Yaskawa INFORM job: KRIS7.JBI

/JOB
//NAME KRIS7
//POS
///NPOS 416,416,416,15,0,0
///TOOL 0
///POSTYPE PULSE
///PULSE
C00000=-36471,-76527,-106813,19264,71481,77238
C00001=-36471,-76527,-106813,19264,71481,77238
C00002=-63812,-119516,-80644,-27282,71106,59809
C00003=-86670,-29465,-24103,-33182,93398,46515
C00004=-88663,-31189,-25266,-33292,92471,45985
C00005=-89600,-31952,-25776,-33339,92036,45737
C00006=-88663,-31189,-25266,-33292,92471,45985
C00007=-88663,-31929,-28188,-33361,93666,45629
C00008=-101397,-33118,-34088,-22474,91022,41668
C00009=-101397,-32934,-33069,-22469,90527,41762
C00010=-101397,-33275,-35023,-22483,91481,41581
C00011=-104499,20623,14787,-23283,115207,62973
C00012=-104352,17765,12486,-23220,115200,63034
C00013=-104529,15851,10717,-23303,115245,62949
C00014=-104352,17765,12486,-23220,115200,63034
C00015=-100086,19810,13187,-22516,115799,63398
C00016=-93288,781,-1160,-33549,91987,44264
C00017=-95103,1586,-482,-33591,91265,43744
C00018=-95638,1156,-842,-33600,91054,43591
C00019=-95103,1586,-482,-33591,91265,43744
C00020=-100253,-3614,-11898,-25466,91372,41970
C00021=-107199,-8537,-17665,-19004,89460,40114
C00022=-108350,-8919,-17473,-17740,88760,39873
C00023=-102096,-5783,-13006,-25389,90415,41488
C00024=-93175,-13453,-24658,-25770,96080,43586
C00025=-29596,-126908,-80456,-16683,91164,67663
C00026=-130966,-130992,-81417,14801,93022,-34731
C00027=-139735,-123676,-71676,23223,79574,-40827
C00028=-136755,-124231,-71804,23689,78586,-39979
C00029=-134984,-124514,-71869,23951,78010,-39473
C00030=-136755,-124231,-71804,23689,78586,-39979
C00031=-136306,-124758,-74432,23664,79703,-39597
C00032=-105195,-127447,-79852,15126,73259,-28242
C00033=-104798,-126140,-77647,15190,72530,-28198
C00034=-108375,-128078,-79564,15067,73342,-29336
C00035=-112121,-93277,-65445,16297,96104,-47809
C00036=-116095,-84503,-58814,18813,102506,-48434
C00037=-114391,-86924,-59797,19239,101506,-47972
C00038=-116095,-84503,-58814,18813,102506,-48434
C00039=-117812,-129995,-81150,14641,74986,-32390
C00040=-118791,-92886,-67151,14205,85296,-31516
C00041=-116748,-92781,-67110,14299,84968,-30842
C00042=-115499,-92681,-67072,14351,84774,-30431
C00043=-116748,-92781,-67110,14299,84968,-30842
C00044=-116748,-94243,-70296,14285,86141,-30707
C00045=-102870,-92009,-70676,9222,86435,-25689
C00046=-102870,-90997,-68303,9229,85506,-25758
C00047=-102870,-92009,-70676,9222,86435,-25689
C00048=-124106,-98193,-79828,8318,91183,-32632
C00049=-120990,-117719,-86799,1028,78019,83969
C00050=-103618,-122878,-84450,6731,45671,69045
C00051=-107839,-39273,-43881,11021,86771,60654
C00052=-102663,-26959,-34255,5037,90909,61236
C00053=-106417,-22492,-30421,10624,98396,60708
C00054=-103076,-37240,-40581,8849,97261,61678
C00055=-110992,-39766,-43585,17340,97602,59383
C00056=-111851,-103912,-94699,10334,87868,68255
C00057=-100525,-93554,-87313,9422,87254,72087
C00058=-95765,-72558,-76889,7644,100510,59309
C00059=-95463,-76426,-71939,16938,115118,61391
C00060=-102124,-64154,-61473,23072,122501,60539
C00061=-108072,-63754,-61449,27079,123073,58329
C00062=-126453,-110744,-88068,25157,96958,85114
C00063=-124535,-114305,-86499,25277,93833,85163
C00064=-121951,-112497,-85625,25654,93398,86032
C00065=-116232,-108405,-84002,26384,92604,88006
C00066=-122754,-106725,-87203,25770,97209,86568
C00067=-142865,-91008,-85242,17891,113758,73123
C00068=-142005,-90205,-84914,18160,113770,73464
C00069=-93871,-48257,-54590,-14207,101968,-48555
C00070=-106716,17042,-5346,-15024,102835,-53222
C00071=-114740,-14345,-34597,-13608,101053,-59815
C00072=-127078,-3386,-21930,-8482,103399,-53955
C00073=-129021,-1243,-17298,-7607,102543,-53064
C00074=-129893,-13096,-22178,-14005,113849,-54571
C00075=-129597,-5294,-13720,-15224,118044,-55057
C00076=-122058,-3228,-13278,-23261,119236,-52777
C00077=-102997,28917,14853,-20600,116287,-84527
C00078=-102792,-6395,-13177,-23260,105514,-87254
C00079=-105472,-3384,-9862,-23514,105257,-88219
C00080=-107060,-2107,-8876,-23770,104848,-88744
C00081=-104416,1445,-8009,-23523,106791,-88129
C00082=-100743,5943,-9423,-11985,113108,-51981
C00083=-104100,-22795,-28366,-25068,61310,-50210
C00084=-122112,-33809,-21710,-17217,45375,-58941
C00085=-130767,-31374,-20493,-827,48037,-55558
C00086=-127443,-25046,-15801,-6227,47707,-53970
C00087=-124818,-6385,-1356,-9028,48013,-52772
C00088=-117469,-7945,-6130,-22808,51414,-49873
C00089=-27812,-119319,-87277,-42007,83182,-24370
C00090=-5621,-139291,-109992,-39952,96377,80222
C00091=-5621,-139291,-109992,-39952,96377,80222
C00092=87039,-115654,-82424,8022,52039,63522
C00093=129513,-144814,-136934,9080,53426,64546
C00094=129513,-144814,-136934,9080,53426,64546
C00095=129513,-109632,-69732,14359,30578,61412
C00096=129513,-83278,-28536,22379,19314,57484
C00097=122399,-55102,-4999,-8402,35911,61097
C00098=119920,-45288,5620,-7331,30390,60229
C00099=119750,-46058,4611,-7150,30605,60108
C00100=119750,-45110,6218,-7257,30106,60163
C00101=119736,-46268,4531,-7151,30546,60106
C00102=119736,-47260,4985,-7320,29764,60193
C00103=119733,-47115,5156,-7324,29732,60195
C00104=119739,-46062,5830,-7299,29854,60181
C00105=119715,-47768,4014,-7231,30094,60141
C00106=122330,-55612,-6297,-8657,32618,61353
C00107=121709,-73745,-24049,9098,30676,53116
C00108=129398,-114812,-46545,3278,22913,57364
C00109=129398,-114812,-46545,3278,22913,57364
C00110=147189,-126166,-80752,5474,34460,60082
C00111=165214,-137669,-115409,7698,46160,62836
C00112=176409,-144814,-136934,9080,53426,64546
C00113=176409,-109327,-69248,14418,30440,61382
C00114=137996,-109327,-69248,14418,30440,61382
C00115=136854,5077,41656,21727,21645,57624
C00116=123203,14789,51546,53172,38991,40073
C00117=123077,34948,78392,59944,35543,36223
C00118=123077,37993,83408,61838,34770,35183
C00119=123098,35348,79007,60153,35442,36112
C00120=123139,31348,74887,59568,35673,36443
C00121=123149,34907,80133,61289,34946,35499
C00122=123130,37074,82445,61677,34805,35280
C00123=123183,30422,73312,58971,35912,36781
C00124=123599,57381,99984,51632,43856,40437
C00125=128629,59731,102899,52063,41097,41453
C00126=130023,30320,69348,52154,35987,38987
C00127=132104,19481,50493,23737,37003,47692
C00128=136200,48792,78585,9333,46433,53780
C00129=127667,43842,73216,11867,48213,50363
C00130=127110,36942,61073,12684,52130,50324
C00131=125174,17943,48073,21449,38985,45601
C00132=109988,7135,45797,56276,48109,34557
C00133=110783,-2370,26113,10588,43916,42309
C00134=96618,15106,36280,16308,48845,36588
C00135=99195,57631,83562,8929,54990,39222
C00136=83229,75338,108095,18392,45531,30732
C00137=82057,52050,70954,17595,54461,31693
C00138=99279,-29834,2408,12633,51480,38376
C00139=124602,-34297,-476,3581,48489,48797
C00140=129000,-155474,-110821,1722,53982,50766
C00141=129000,-186332,-136923,1718,54189,50769
C00142=129000,-186332,-136923,1718,54189,50769
C00143=124634,-42983,-17396,3288,54424,49011
C00144=119975,43106,65207,5416,48088,46799
C00145=124227,21838,45287,-4126,60993,49348
C00146=115102,22260,45694,-2630,60591,46004
C00147=111900,23179,46586,-2094,60423,44829
C00148=106599,25422,48781,-1196,60121,42879
C00149=109500,51617,73450,-2873,46958,44240
C00150=119708,-19564,1692,5024,54962,47046
C00151=124398,4257,31803,38326,49723,41965
C00152=124500,-5455,16693,36249,53145,43496
C00153=123978,22175,41893,32824,63757,46964
C00154=136633,26599,46213,31259,58773,50852
C00155=137127,47274,64261,33367,46328,47205
C00156=127043,-60461,-47717,31537,61680,47716
C00157=130427,-104246,-66216,34447,50964,45598
C00158=130427,-131180,-133049,27346,74705,52630
C00159=129293,-131648,-133187,27764,74930,52255
C00160=129293,-112975,-80869,32941,55210,46617
C00161=125224,-26758,-13299,33226,59088,46051
C00162=97492,-17863,6740,47317,62068,35221
C00163=76763,21057,43225,48272,71101,29312
C00164=80709,51150,75439,39481,73131,33496
C00165=101893,22474,45257,39781,66883,40263
C00166=98002,-1326,18556,46821,62661,35806
C00167=97492,-17863,6740,47317,62068,35221
C00168=125224,-26758,-13299,33226,59088,46051
C00169=129293,-131648,-133187,27764,74930,52255
C00170=129293,-130373,-135142,27565,76585,52657
C00171=129293,-130373,-135142,27565,76585,52657
C00172=129293,-130373,-135142,27565,76585,52657
C00173=126775,-65943,-41926,33631,56357,45828
C00174=146499,-5820,8509,-12483,47348,74367
C00175=133227,18598,33392,-5127,43166,68552
C00176=134087,40556,59352,-4333,44134,68757
C00177=109518,39473,58200,8432,44907,57480
C00178=110804,22133,33080,8574,45677,58038
C00179=95832,-100308,-60228,18401,42759,50383
C00180=85717,-180836,-128237,23276,45701,46095
C00181=134324,-194207,-130804,-6935,34984,69726
C00182=134324,-194207,-130804,-6935,34984,69726
C00183=134324,-194207,-130804,-6935,34984,69726
C00184=126554,-62104,-55568,-768,56192,65237
C00185=102691,-29899,-32559,11070,60126,55987
C00186=93699,-1684,15739,18283,46963,50224
C00187=95177,34388,59282,20423,38809,49091
C00188=95427,37375,44105,11480,58003,52927
C00189=82804,57701,66332,15963,56969,47713
C00190=80078,42075,52490,24500,50349,44630
C00191=92595,-4722,8571,18053,49920,50291
C00192=90890,13188,28851,45241,66990,53478
C00193=96516,51970,78121,48970,56932,51018
C00194=108766,35550,55769,36284,51974,56943
C00195=109501,48300,76470,39344,46724,54946
C00196=112089,47430,75488,38680,45769,55875
C00197=109461,35195,57508,36711,50675,56747
C00198=102961,43860,64049,37370,53600,54832
C00199=117347,37004,56694,33344,48695,60037
C00200=107165,27849,47408,45061,56134,56400
C00201=93699,-1684,15739,18283,46963,50224
C00202=126554,-62104,-55568,-768,56192,65237
C00203=132741,-190295,-136907,-5065,40605,68463
C00204=132741,-190295,-136907,-5065,40605,68463
C00205=132741,-190295,-136907,-5065,40605,68463
C00206=132741,-190295,-136907,-5065,40605,68463
C00207=126216,-48827,-32555,-652,48851,65144
C00208=116157,12397,26645,-836,43828,61032
C00209=107201,15073,29086,4732,43915,56787
C00210=108708,45240,59560,984,53519,57995
C00211=105889,47117,61614,1966,53270,56850
C00212=104117,15965,27840,6481,45345,55424
C00213=116157,12397,26645,-836,43828,61032
C00214=115184,32776,48658,-853,48273,60616
C00215=102009,39914,56094,5283,47719,54846
C00216=104295,38849,56164,-3583,45498,56420
C00217=106773,10666,21679,-1556,45201,57174
C00218=121513,8451,23347,32656,44981,60126
C00219=121325,33244,54124,32762,45132,60075
C00220=136244,38436,59676,26271,39414,66032
C00221=133358,13884,30500,26959,39421,64637
C00222=126216,-48827,-32555,-652,48851,65144
C00223=132741,-190295,-136907,-5065,40605,68463
C00224=132741,-190295,-136907,-5065,40605,68463
C00225=132741,-190295,-136907,-5065,40605,68463
C00226=132741,-190295,-136907,-5065,40605,68463
C00227=126554,-62104,-55568,-768,56192,65237
C00228=93699,-1684,15739,18283,46963,50224
C00229=109219,22842,33799,17593,55341,60017
C00230=115088,32680,55692,7882,41104,61696
C00231=98115,43367,67193,11592,40390,54327
C00232=92675,33947,50979,20393,49569,52577
C00233=113935,26100,44118,24451,47496,60162
C00234=114558,35388,59860,26260,42851,59091
C00235=117732,34768,59212,24806,41998,60459
C00236=114305,24559,43264,24398,47147,60243
C00237=99844,11402,27037,25299,53213,55440
C00238=126554,-62104,-55568,-768,56192,65237
C00239=132741,-190295,-136907,-5065,40605,68463
C00240=132741,-190295,-136907,-5065,40605,68463
C00241=132741,-190295,-136907,-5065,40605,68463
C00242=132741,-190295,-136907,-5065,40605,68463
C00243=126216,-48827,-32555,-652,48851,65144
C00244=134748,7082,18366,-200,46227,68791
C00245=132038,36511,51354,2924,49864,67481
C00246=110399,36003,50767,11764,51912,58463
C00247=101806,27679,40045,16592,51225,54569
C00248=102258,33237,49963,17192,48019,54198
C00249=104874,31614,48575,4374,45128,56525
C00250=106858,16986,29459,6761,48587,57166
C00251=113156,-2573,6178,11839,50347,59373
C00252=100847,-116604,-69788,21646,41420,51852
C00253=93537,-194381,-130385,26473,40988,47897
C00254=104459,-185785,-128899,13362,14722,54877
C00255=137185,-168918,-120422,-22616,31853,56508
C00256=103466,-143035,-89833,18127,44217,-664
C00257=153034,-42791,-3789,-574,51224,21077
C00258=154411,-23786,22188,6392,45845,11810
C00259=163692,-14831,30793,3045,43978,15753
C00260=162658,-12144,32796,3380,44162,15317
C00261=162658,-10372,35929,3443,43146,15280
C00262=162658,-10822,35136,3427,43403,15291
C00263=163644,-13399,33193,3102,43239,15709
C00264=163644,-12612,34572,3127,42795,15690
C00265=163043,-11060,35746,3327,42891,15434
C00266=163515,-12286,34819,3170,42815,15635
C00267=166152,-32133,5550,1997,50546,16952
C00268=100006,-46830,-3879,17345,57754,-8477
C00269=55652,-4276,24712,7053,56203,-22524
C00270=50070,19037,58848,16400,45172,-27179
C00271=51341,29328,71603,16783,42484,-27133
C00272=51341,32600,77102,17341,40853,-27469
C00273=51341,31422,75137,17137,41430,-27347
C00274=50264,28853,72458,17349,41942,-27728
C00275=50264,30492,75208,17635,41129,-27900
C00276=50738,31631,76404,17545,40896,-27733
C00277=50419,30858,75590,17605,41054,-27844
C00278=50419,14018,45638,14959,50461,-26136
C00279=53903,-12653,21571,13778,50962,-24612
C00280=66094,-67687,-18476,10677,45688,-20127
C00281=87454,-109874,-47340,-27972,40441,7116
C00282=78946,-55292,-6224,-23492,40558,2756
C00283=70027,-40972,10385,-20890,35738,-464
C00284=63439,-31094,22495,-18522,32104,-3061
C00285=63439,-29243,25592,-19018,31198,-2801
C00286=75556,-28394,37292,-62320,27769,16956
C00287=74155,-27422,37887,-61985,27131,16453
C00288=64318,-30449,24372,-21159,31089,-1672
C00289=67917,-25293,27676,-22824,32488,-51
C00290=67917,-25293,27676,-22824,32488,-51
C00291=68696,-24050,28500,-23162,32795,289
C00292=67917,-25293,27676,-22824,32488,-51
C00293=75368,-51805,-10970,-21451,43738,562
C00294=86139,-25078,5298,-24076,50017,4008
C00295=83917,-18337,16451,-24570,46284,3982
C00296=79836,-11066,25880,-23931,43276,2865
C00297=79836,-9413,28995,-24399,42297,3151
C00298=86314,-11086,32289,-42271,40319,10375
C00299=84998,-9998,33124,-41890,39785,9892
C00300=80963,-11349,26642,-26884,42529,4054
C00301=82363,-6834,30155,-27320,43093,4575
C00302=82761,-5465,31244,-27447,43243,4725
C00303=83186,-3958,32457,-27584,43396,4888
C00304=82761,-5465,31244,-27447,43243,4725
C00305=87385,-23200,183,-25112,53654,3858
C00306=88611,-6659,17671,-26227,51974,4862
C00307=85936,239,26154,-25964,49655,4281
C00308=85936,1480,28752,-26325,48787,4530
C00309=91127,630,32748,-40408,46738,9768
C00310=90313,1326,33333,-40211,46382,9497
C00311=86792,7,26768,-28149,49107,5083
C00312=90602,-33059,-4237,-28517,52203,5912
C00313=94576,-67258,-23025,57506,77870,-531
C00314=122383,-58832,-3556,65417,58097,774
C00315=127343,-13643,25366,63114,57669,4189
C00316=131296,13324,53885,65824,53660,3026
C00317=131296,14618,56173,66322,53341,2642
C00318=130824,14275,55697,67245,54004,2465
C00319=131723,14569,55971,67399,53464,2593
C00320=130860,14268,55674,67244,53987,2476
C00321=127124,-5804,29633,63377,58737,4694
C00322=126701,-15037,22522,63119,61223,3769
C00323=126701,1136,51385,68187,57095,-774
C00324=131284,6353,59362,70779,53649,-1335
C00325=131284,8754,63319,71617,53230,-1977
C00326=131284,6353,59362,70779,53649,-1335
C00327=132452,6685,59657,71098,52984,-1198
C00328=131284,6353,59362,70779,53649,-1335
C00329=131052,11501,64001,70861,53706,-1474
C00330=130893,14100,66417,70922,53742,-1574
C00331=130719,17099,69269,71021,53763,-1708
C00332=130893,14100,66417,70922,53742,-1574
C00333=128315,-22064,27147,66784,57381,941
C00334=129627,-37207,17556,68184,55855,186
C00335=130148,-23471,44300,74760,52317,-4741
C00336=135320,-14449,56479,79067,48853,-5949
C00337=135320,-12066,60154,79963,48630,-6563
C00338=135320,-14449,56479,79067,48853,-5949
C00339=137070,-14043,56767,79770,47945,-5809
C00340=135320,-14449,56479,79067,48853,-5949
C00341=134716,-10676,59212,78597,49226,-5841
C00342=134466,-8976,60486,78417,49378,-5807
C00343=134182,-6930,62050,78227,49545,-5776
C00344=134466,-8976,60486,78417,49378,-5807
C00345=106496,-51026,-9475,59829,73743,881
C00346=106496,-62277,-31108,58328,77765,3910
C00347=137468,-45448,-13164,23993,62707,9546
C00348=142031,-34381,-3630,18745,59946,9254
C00349=153480,-23481,18954,7895,48240,10284
C00350=154576,-15419,32985,7624,43640,10304
C00351=154522,-15140,33190,7639,43662,10282
C00352=163868,-10589,37972,6252,39486,12143
C00353=163705,-4288,45034,21073,38117,2051
C00354=163923,-2936,48273,26703,35302,170
C00355=146970,-27557,19782,29282,44621,-5055
C00356=77984,-28544,12598,9594,52255,-4511
C00357=87028,-14899,33509,-8097,43242,2023
C00358=86974,-14913,33498,-8080,43236,2001
C00359=77485,-7266,39372,-4959,42873,-2067
C00360=74579,-2521,47308,-17915,35684,548
C00361=75615,102,52227,-26296,32839,3633
C00362=84696,-19604,28451,-27180,39406,6073
C00363=87454,-109874,-47340,-27972,40441,7116
C00364=87454,-109874,-47340,-27972,40441,7116
C00365=73980,-36973,3355,-18473,60366,27525
C00366=58877,-27993,19766,-16405,50257,19650
C00367=71120,-6285,35203,-17245,53240,22132
C00368=69479,-8808,33067,-14788,50723,16894
C00369=73605,-31096,1389,-14177,59206,17320
C00370=72431,-18207,17991,-16956,51529,14828
C00371=73562,-15726,19761,-17396,52120,15565
C00372=83313,14185,44247,-21039,56473,22237
C00373=84211,-11070,13701,-18734,53182,26231
C00374=82998,-523,24465,-18637,51768,25979
C00375=82448,-570,28041,-15362,40529,26924
C00376=77134,-2165,39833,11119,14146,19838
C00377=76844,-12553,31864,7458,12108,20601
C00378=84341,-54767,463,-16268,10060,32559
C00379=79893,-46463,9240,-49361,8484,37720
C00380=71243,-22477,30789,30336,5200,-490
C00381=70979,-19028,33557,31433,5346,-1026
C00382=68683,-10375,50772,112552,4351,-37626
C00383=72976,-34040,25530,30096,2440,-170
C00384=51638,-47354,18402,88201,13764,-30312
C00385=50365,-30767,37744,101133,14655,-36527
C00386=46532,-17600,60099,119714,18815,-46088
C00387=50533,-52861,21550,106572,14840,-38992
C00388=66288,-93178,-46103,5866,60369,16168
C00389=112510,-98188,-44790,18471,62864,-44268
C00390=149625,-37879,6780,17046,57011,-35751
C00391=155605,-32525,16928,15112,50177,-29308
C00392=149418,-7594,34122,13784,51545,-27133
C00393=143716,-10385,36525,25765,46016,-27057
C00394=147766,-22217,9496,11268,57983,-23560
C00395=146875,-12758,20894,15319,55227,-24771
C00396=146053,-8471,24161,15451,55560,-25047
C00397=142035,19351,48051,16301,55907,-26583
C00398=141803,14161,44980,18392,51510,-21349
C00399=142040,5818,24378,13474,61789,-22474
C00400=138840,15265,37176,20739,58625,-24937
C00401=138706,17261,38894,20771,58629,-24991
C00402=139526,10572,40705,23596,37058,-29346
C00403=140566,11430,47120,26457,25355,-31911
C00404=140419,-8993,28489,25719,26277,-31573
C00405=142059,-17553,21658,25375,25949,-31323
C00406=143624,-11159,28730,24740,24544,-30775
C00407=144392,-5853,43056,31020,18891,-33660
C00408=150093,-42733,14524,24992,16002,-29807
C00409=146967,-32270,24662,40502,20136,-34953
C00410=144755,-20255,35089,33636,31779,-30408
C00411=144236,-61611,5153,41773,14596,-38681
C00412=136995,-150356,-85047,33892,64386,-36535
C00413=136995,-178339,-110283,33604,8697,-36217
C00414=130728,-161100,-136081,16173,33339,-28558
C00415=1271,-161100,-136081,16173,33339,-28558
BC00000=295325,674563,1075170
BC00001=295325,674563,1075170
BC00002=396971,731967,797664
BC00003=396971,731967,797664
BC00004=396971,731967,797664
BC00005=396971,731967,797664
BC00006=396971,731967,797664
BC00007=396971,731967,797664
BC00008=396971,731967,797664
BC00009=396971,731967,797664
BC00010=396971,731967,797664
BC00011=396971,731967,797664
BC00012=396971,731967,797664
BC00013=396971,731967,797664
BC00014=396971,731967,797664
BC00015=396971,731967,797664
BC00016=396971,731967,797664
BC00017=396971,731967,797664
BC00018=396971,731967,797664
BC00019=396971,731967,797664
BC00020=396971,731967,797664
BC00021=396971,731967,797664
BC00022=396971,731967,797664
BC00023=396971,731967,797664
BC00024=396971,731967,797664
BC00025=396971,731967,797664
BC00026=1331,731967,797664
BC00027=1331,834817,797664
BC00028=1331,834817,797664
BC00029=1331,834817,797664
BC00030=1331,834817,797664
BC00031=1331,834817,797664
BC00032=1331,834817,797664
BC00033=1331,834817,797664
BC00034=1331,834817,797664
BC00035=1331,834817,797664
BC00036=1331,834817,797664
BC00037=1331,834817,797664
BC00038=1331,834817,797664
BC00039=1331,834817,797664
BC00040=1331,834817,797664
BC00041=1331,834817,797664
BC00042=1331,834817,797664
BC00043=1331,834817,797664
BC00044=1331,834817,797664
BC00045=1331,834817,797664
BC00046=1331,834817,797664
BC00047=1331,834817,797664
BC00048=1331,834817,797664
BC00049=1072,761065,516765
BC00050=1072,827865,516765
BC00051=1071,829671,517043
BC00052=1071,829895,517078
BC00053=1071,829895,517078
BC00054=1071,829895,517078
BC00055=1071,829895,517078
BC00056=768,829895,695080
BC00057=768,829895,695080
BC00058=768,829895,695080
BC00059=768,829895,695080
BC00060=768,829895,695080
BC00061=768,829895,695080
BC00062=768,829895,695080
BC00063=768,829895,695080
BC00064=768,829895,695080
BC00065=768,829895,695080
BC00066=768,829895,695080
BC00067=768,829895,695080
BC00068=768,686767,695080
BC00069=396971,681851,797664
BC00070=396971,731967,797664
BC00071=396971,731967,797664
BC00072=396971,731967,797664
BC00073=396971,731967,797664
BC00074=396971,731967,797664
BC00075=396971,731967,797664
BC00076=396971,731967,797664
BC00077=396971,731967,797664
BC00078=396971,731967,797664
BC00079=396971,731967,797664
BC00080=396971,731967,797664
BC00081=396971,731967,797664
BC00082=396971,731967,797664
BC00083=396971,731967,516765
BC00084=396971,731967,516765
BC00085=396971,731967,516765
BC00086=396972,731979,516765
BC00087=396971,731967,516765
BC00088=396971,731967,516765
BC00089=396971,731967,516765
BC00090=188286,731967,1013423
BC00091=188286,774486,1052805
BC00092=125948,1177450,1071719
BC00093=215453,1309115,984509
BC00094=345399,1357897,984509
BC00095=345399,1357897,984509
BC00096=345399,1230997,984509
BC00097=346767,1230997,984506
BC00098=346767,1230997,984506
BC00099=346767,1230997,984506
BC00100=346767,1230997,984506
BC00101=346767,1230997,984506
BC00102=346767,1230997,984506
BC00103=346767,1230997,984506
BC00104=346767,1230997,984506
BC00105=346767,1230997,984506
BC00106=346767,1230997,984506
BC00107=309515,1253158,984507
BC00108=309515,1253158,984507
BC00109=309515,1328360,1051553
BC00110=314470,1361455,1064018
BC00111=253389,1357693,1050986
BC00112=215453,1309115,984509
BC00113=215453,1309115,984509
BC00114=135997,1309115,984509
BC00115=135997,1309115,984509
BC00116=135997,1309115,984509
BC00117=135997,1309115,984505
BC00118=135997,1309115,984505
BC00119=135997,1309115,984505
BC00120=135997,1309115,984505
BC00121=135997,1309115,984505
BC00122=135997,1309115,984505
BC00123=135997,1309115,984505
BC00124=135997,1309115,984509
BC00125=135997,1309115,984509
BC00126=135997,1309115,984509
BC00127=135997,1309115,984509
BC00128=135997,1309115,984509
BC00129=135997,1309115,984509
BC00130=135997,1309115,984509
BC00131=135997,1309115,984509
BC00132=135997,1309115,984509
BC00133=135997,1309115,984509
BC00134=94463,1309115,955550
BC00135=94463,1309115,963176
BC00136=94463,1309115,963176
BC00137=94463,1309115,963176
BC00138=94463,1309115,963176
BC00139=141941,1309115,963176
BC00140=141941,1309115,963176
BC00141=223116,1330631,963176
BC00142=328548,1330631,963176
BC00143=328548,1330631,963176
BC00144=328548,1330631,963176
BC00145=328548,1285890,963176
BC00146=328548,1285890,963176
BC00147=328548,1285890,963176
BC00148=328548,1285890,963176
BC00149=328548,1330631,963176
BC00150=328548,1291307,959498
BC00151=328548,1293601,963176
BC00152=328548,1288886,905196
BC00153=328548,1288886,905196
BC00154=328548,1288886,905196
BC00155=328824,1330631,905196
BC00156=328824,1330631,905196
BC00157=328824,1330631,905196
BC00158=328824,1330631,905196
BC00159=151003,1330631,905196
BC00160=151003,1330631,905196
BC00161=151003,1330631,905196
BC00162=103648,1289163,905196
BC00163=103648,1289163,905196
BC00164=103648,1289163,905196
BC00165=103648,1289163,905196
BC00166=103648,1289163,905196
BC00167=103648,1289163,905196
BC00168=151003,1330631,905196
BC00169=151003,1330631,905196
BC00170=151003,1330631,905196
BC00171=303803,1330631,905196
BC00172=303803,1330631,763831
BC00173=303803,1330631,902112
BC00174=303803,1330631,902112
BC00175=303803,1330631,902112
BC00176=303803,1330631,902112
BC00177=303803,1330631,902112
BC00178=303803,1330631,902112
BC00179=303803,1330631,902112
BC00180=303803,1330631,1003127
BC00181=236612,1330631,1003127
BC00182=137483,1330631,1003127
BC00183=136337,1325904,719417
BC00184=136337,1325904,818715
BC00185=87820,1325904,842743
BC00186=87820,1325904,951848
BC00187=87820,1325904,951848
BC00188=87820,1320020,844218
BC00189=87820,1320020,844218
BC00190=87820,1325904,927335
BC00191=87820,1325904,927335
BC00192=87820,1325904,927335
BC00193=87820,1325904,927335
BC00194=87820,1325904,927335
BC00195=87820,1325904,927335
BC00196=87820,1325904,927335
BC00197=87820,1325904,927335
BC00198=87820,1325904,890762
BC00199=87820,1325904,890392
BC00200=87820,1325904,927335
BC00201=87820,1325904,951848
BC00202=136337,1325904,818715
BC00203=136337,1325904,818715
BC00204=136337,1325904,998300
BC00205=310720,1325904,998300
BC00206=310720,1325904,777065
BC00207=310720,1325904,891809
BC00208=310720,1325904,891809
BC00209=310720,1325904,891809
BC00210=310720,1325904,891809
BC00211=310720,1325904,891809
BC00212=310720,1325904,891809
BC00213=310720,1325904,891809
BC00214=310720,1325904,891809
BC00215=310720,1325904,891809
BC00216=310720,1325904,891809
BC00217=310720,1325904,891809
BC00218=310720,1325904,891809
BC00219=310720,1325904,891809
BC00220=310720,1325904,891809
BC00221=310720,1325904,891809
BC00222=310720,1325904,891809
BC00223=310720,1325904,777065
BC00224=310720,1325904,998300
BC00225=136337,1325904,998300
BC00226=136337,1325904,818715
BC00227=136337,1325904,818715
BC00228=87820,1325904,951848
BC00229=87820,1325904,927335
BC00230=87820,1325904,927335
BC00231=87820,1325904,927335
BC00232=87820,1325904,927335
BC00233=87820,1325904,927335
BC00234=87820,1325904,927335
BC00235=87820,1325904,927335
BC00236=87820,1325904,927335
BC00237=87820,1325904,927335
BC00238=136337,1325904,818715
BC00239=136337,1325904,818715
BC00240=136337,1325904,998300
BC00241=310720,1325904,998300
BC00242=310720,1325904,777065
BC00243=310720,1325904,891809
BC00244=310720,1325904,891809
BC00245=310720,1325904,891809
BC00246=310720,1325904,891809
BC00247=310720,1325904,891809
BC00248=310720,1325904,891809
BC00249=310720,1325904,891809
BC00250=310720,1325904,891809
BC00251=310720,1325904,891809
BC00252=310720,1325904,891809
BC00253=310720,1325904,1051225
BC00254=230237,1331507,1051225
BC00255=214487,1257960,1051225
BC00256=187930,1133951,1051225
BC00257=187930,1063861,1051225
BC00258=187930,1063861,1051225
BC00259=187931,1063862,1051199
BC00260=187931,1063862,1051199
BC00261=187931,1063862,1051199
BC00262=187931,1063862,1051199
BC00263=187931,1063862,1051199
BC00264=187931,1063862,1051199
BC00265=187931,1063862,1051199
BC00266=187931,1063862,1051199
BC00267=187931,1063862,1051199
BC00268=187930,1063861,1051225
BC00269=187930,1063861,1051225
BC00270=187930,1063861,1051225
BC00271=187930,1063861,1051225
BC00272=187930,1063861,1051225
BC00273=187930,1063861,1051225
BC00274=187930,1063861,1051225
BC00275=187930,1063861,1051225
BC00276=187930,1063861,1051225
BC00277=187930,1063861,1051225
BC00278=187930,1063861,1051225
BC00279=187930,1063861,1051225
BC00280=187930,1063861,1051225
BC00281=244084,1125149,1051225
BC00282=244084,1125149,1051225
BC00283=244084,1125149,1051225
BC00284=244084,1125149,1051225
BC00285=244084,1125149,1051225
BC00286=244084,1125149,1051225
BC00287=244084,1125149,1051225
BC00288=244084,1125149,1051225
BC00289=244084,1125149,1051225
BC00290=244084,1125149,1051225
BC00291=244084,1125149,1051225
BC00292=244084,1125149,1051225
BC00293=244084,1125149,1051225
BC00294=244084,1125149,1051225
BC00295=244084,1125149,1051225
BC00296=244084,1125149,1051225
BC00297=244084,1125149,1051225
BC00298=244084,1125149,1051225
BC00299=244084,1125149,1051225
BC00300=244084,1125149,1051225
BC00301=244084,1125149,1051225
BC00302=244084,1125149,1051225
BC00303=244084,1125149,1051225
BC00304=244084,1125149,1051225
BC00305=244084,1125149,1051225
BC00306=244084,1125149,1051225
BC00307=244083,1125149,1051222
BC00308=244083,1125149,1051222
BC00309=244083,1125149,1051222
BC00310=244083,1125149,1051222
BC00311=244083,1125149,1051222
BC00312=244083,1125149,1051222
BC00313=244083,1125148,1051219
BC00314=166173,1125148,1051219
BC00315=166173,1125148,1051219
BC00316=166173,1142192,1051219
BC00317=166173,1142192,1051219
BC00318=166173,1142192,1051219
BC00319=166173,1142192,1051219
BC00320=166173,1142192,1051219
BC00321=166173,1142192,1051219
BC00322=166173,1142192,1051219
BC00323=166173,1142192,1051219
BC00324=166173,1142192,1051219
BC00325=166173,1142192,1051219
BC00326=166173,1142192,1051219
BC00327=166173,1142192,1051219
BC00328=166173,1142192,1051219
BC00329=166173,1142192,1051219
BC00330=166173,1142192,1051219
BC00331=166173,1142192,1051219
BC00332=166173,1142192,1051219
BC00333=166173,1142192,1051219
BC00334=166173,1142192,1051219
BC00335=166173,1142192,1051219
BC00336=166173,1142192,1051219
BC00337=166173,1142192,1051219
BC00338=166173,1142192,1051219
BC00339=166173,1142192,1051219
BC00340=166173,1142192,1051219
BC00341=166173,1142192,1051219
BC00342=166173,1142192,1051219
BC00343=166173,1142192,1051219
BC00344=166173,1142192,1051219
BC00345=166173,1142192,1051219
BC00346=166173,1142192,1051219
BC00347=180177,1091773,1051223
BC00348=182943,1081815,1051224
BC00349=187709,1064658,1051225
BC00350=187930,1063861,1051225
BC00351=187930,1063861,1051225
BC00352=187930,1063861,1051225
BC00353=187930,1063861,1051225
BC00354=187930,1063861,1051225
BC00355=187930,1063861,1051225
BC00356=244084,1063861,1051225
BC00357=244084,1063861,1051225
BC00358=244084,1063861,1051225
BC00359=244084,1063861,1051225
BC00360=244084,1063861,1051225
BC00361=244084,1063861,1051225
BC00362=244084,1063861,1051225
BC00363=244084,1063861,1051225
BC00364=244084,1125149,1051225
BC00365=244084,1125149,1051225
BC00366=244084,1125149,1051225
BC00367=244084,1125149,1051225
BC00368=244084,1125149,1051225
BC00369=244084,1125149,1051225
BC00370=244084,1125149,1051225
BC00371=244084,1125149,1051225
BC00372=244084,1125149,1051225
BC00373=244084,1125149,1051225
BC00374=244084,1125149,1051225
BC00375=244084,1125149,1051225
BC00376=244084,1125149,1051225
BC00377=244084,1125149,1051225
BC00378=244084,1125149,1051225
BC00379=244084,1125149,1051225
BC00380=244084,1125149,1051225
BC00381=244084,1125149,1051222
BC00382=244084,1125149,1051225
BC00383=244084,1125149,1051225
BC00384=244084,1125149,1051225
BC00385=244083,1125149,1051223
BC00386=244084,1125149,1051225
BC00387=244084,1125149,1051225
BC00388=244084,1125149,1051225
BC00389=148492,1125149,1051225
BC00390=148492,1157650,1055882
BC00391=148492,1157650,1055882
BC00392=148492,1157650,1055882
BC00393=148493,1157650,1055879
BC00394=148492,1157650,1055882
BC00395=148492,1157650,1055882
BC00396=148492,1157650,1055882
BC00397=148492,1157650,1055882
BC00398=148492,1157650,1055882
BC00399=148492,1157650,1055882
BC00400=148492,1157650,1055882
BC00401=148492,1157650,1055882
BC00402=148492,1157650,1055881
BC00403=148492,1157650,1055882
BC00404=148492,1157650,1055882
BC00405=148492,1157650,1055882
BC00406=148492,1157650,1055882
BC00407=148492,1157650,1055882
BC00408=148492,1157650,1055882
BC00409=148492,1157650,1055882
BC00410=148492,1157650,1055882
BC00411=148492,1157650,1055882
BC00412=148492,1157650,1055882
BC00413=189366,1229859,1070827
BC00414=189366,1118575,1070827
BC00415=189366,734808,1070827
EC00000=0,0
EC00001=-88685,-556476
EC00002=-88685,-556476
EC00003=-88685,-556476
EC00004=-88685,-556476
EC00005=-88685,-556476
EC00006=-88685,-556476
EC00007=-88685,-556476
EC00008=-88685,-556476
EC00009=-88685,-556476
EC00010=-88685,-556476
EC00011=-88685,-556476
EC00012=-88685,-556476
EC00013=-88685,-556476
EC00014=-88685,-556476
EC00015=-88685,-556476
EC00016=-88685,-556476
EC00017=-88685,-556476
EC00018=-88685,-556476
EC00019=-88685,-556476
EC00020=-88685,-556476
EC00021=-88685,-556476
EC00022=-88685,-556476
EC00023=-88685,-556476
EC00024=-88685,-556476
EC00025=-88685,-556476
EC00026=-88685,-556476
EC00027=-88685,-556476
EC00028=-88685,-556476
EC00029=-88685,-556476
EC00030=-88685,-556476
EC00031=-88685,-556476
EC00032=-88685,-556476
EC00033=-88685,-556476
EC00034=-88685,-556476
EC00035=-88685,-556476
EC00036=-88685,-556476
EC00037=-88685,-556476
EC00038=-88685,-556476
EC00039=-88685,-556476
EC00040=-88685,-556476
EC00041=-88685,-556476
EC00042=-88685,-556476
EC00043=-88685,-556476
EC00044=-88685,-556476
EC00045=-88685,-556476
EC00046=-88685,-556476
EC00047=-88685,-556476
EC00048=-88685,-556476
EC00049=264893,-556476
EC00050=264893,-556476
EC00051=264346,-556476
EC00052=264278,-556476
EC00053=264278,-556476
EC00054=264278,-556476
EC00055=264278,-556476
EC00056=-85879,-556476
EC00057=-85879,-556476
EC00058=-85879,-556476
EC00059=-85879,-556476
EC00060=-85879,-556476
EC00061=-85879,-556476
EC00062=-85879,-556476
EC00063=-85879,-556476
EC00064=-85879,-556476
EC00065=-85879,-556476
EC00066=-85879,-556476
EC00067=-85879,-556476
EC00068=-85879,-556476
EC00069=-88685,-556476
EC00070=-88685,-556476
EC00071=-88685,-612042
EC00072=-88685,-612042
EC00073=-88685,-612042
EC00074=-88685,-612042
EC00075=-88685,-612042
EC00076=-88685,-612042
EC00077=-88685,-556476
EC00078=-88685,-556476
EC00079=-88685,-556476
EC00080=-88685,-556476
EC00081=-88685,-556476
EC00082=-88685,-556476
EC00083=264893,-556476
EC00084=264893,-605076
EC00085=264893,-605076
EC00086=264894,-605076
EC00087=264893,-605076
EC00088=264893,-605076
EC00089=264893,-556476
EC00090=264890,-556476
EC00091=264890,-556476
EC00092=-210078,-556477
EC00093=-270405,-556477
EC00094=-270405,-556477
EC00095=-270405,-556477
EC00096=-270405,-556477
EC00097=-270404,-556477
EC00098=-270404,-556477
EC00099=-270404,-556477
EC00100=-270404,-556477
EC00101=-270404,-556477
EC00102=-270404,-556477
EC00103=-270404,-556477
EC00104=-270404,-556477
EC00105=-270404,-556477
EC00106=-270404,-556477
EC00107=-270404,-556477
EC00108=-270404,-556477
EC00109=-270404,-556477
EC00110=-270404,-556477
EC00111=-270405,-556477
EC00112=-270405,-556477
EC00113=-270405,-556477
EC00114=-270405,-556477
EC00115=-270405,-556477
EC00116=-270405,-556477
EC00117=-270404,-556477
EC00118=-270404,-556477
EC00119=-270404,-556477
EC00120=-270404,-556477
EC00121=-270404,-556477
EC00122=-270404,-556477
EC00123=-270404,-556477
EC00124=-270405,-556477
EC00125=-270405,-556477
EC00126=-270405,-556477
EC00127=-270405,-556477
EC00128=-270405,-556477
EC00129=-270405,-556477
EC00130=-270405,-556477
EC00131=-270405,-556477
EC00132=-270405,-556477
EC00133=-270405,-556477
EC00134=-270405,-556477
EC00135=-270405,-556477
EC00136=-270405,-556477
EC00137=-270405,-556477
EC00138=-270405,-556477
EC00139=-270405,-556477
EC00140=-270405,-556477
EC00141=-270405,-556477
EC00142=-270405,-556477
EC00143=-270405,-556477
EC00144=-270405,-556477
EC00145=-270405,-556477
EC00146=-270405,-556477
EC00147=-270405,-556477
EC00148=-270405,-556477
EC00149=-270405,-556477
EC00150=-270405,-556477
EC00151=-270405,-556477
EC00152=-270405,-556477
EC00153=-270405,-556477
EC00154=-270405,-556477
EC00155=-270405,-556477
EC00156=-270405,-556477
EC00157=-270405,-556477
EC00158=-270405,-556477
EC00159=-270405,-556477
EC00160=-270405,-556477
EC00161=-270405,-556477
EC00162=-270405,-556477
EC00163=-270405,-556477
EC00164=-270405,-556477
EC00165=-270405,-556477
EC00166=-270405,-556477
EC00167=-270405,-556477
EC00168=-270405,-556477
EC00169=-270405,-556477
EC00170=-270405,-556477
EC00171=-270405,-556477
EC00172=-270405,-556477
EC00173=-270405,-556477
EC00174=-270405,-556477
EC00175=-270405,-556477
EC00176=-270405,-556477
EC00177=-270405,-556477
EC00178=-270405,-556477
EC00179=-270405,-556477
EC00180=-270405,-556477
EC00181=-270405,-556477
EC00182=-270405,-556477
EC00183=-270405,-556477
EC00184=-270405,-556477
EC00185=-270405,-556477
EC00186=-270405,-556477
EC00187=-270405,-556477
EC00188=-270405,-556477
EC00189=-270405,-556477
EC00190=-270405,-556477
EC00191=-270405,-556477
EC00192=-270405,-556477
EC00193=-270405,-556477
EC00194=-270405,-556477
EC00195=-270405,-556477
EC00196=-270405,-556477
EC00197=-270405,-556477
EC00198=-270405,-556477
EC00199=-270405,-556477
EC00200=-270405,-556477
EC00201=-270405,-556477
EC00202=-270405,-556477
EC00203=-270405,-556477
EC00204=-270405,-556477
EC00205=-270405,-556477
EC00206=-270405,-556477
EC00207=-270405,-556477
EC00208=-270405,-556477
EC00209=-270405,-556477
EC00210=-270405,-556477
EC00211=-270405,-556477
EC00212=-270405,-556477
EC00213=-270405,-556477
EC00214=-270405,-556477
EC00215=-270405,-556477
EC00216=-270405,-556477
EC00217=-270405,-556477
EC00218=-270405,-556477
EC00219=-270405,-556477
EC00220=-270405,-556477
EC00221=-270405,-556477
EC00222=-270405,-556477
EC00223=-270405,-556477
EC00224=-270405,-556477
EC00225=-270405,-556477
EC00226=-270405,-556477
EC00227=-270405,-556477
EC00228=-270405,-556477
EC00229=-270405,-556477
EC00230=-270405,-556477
EC00231=-270405,-556477
EC00232=-270405,-556477
EC00233=-270405,-556477
EC00234=-270405,-556477
EC00235=-270405,-556477
EC00236=-270405,-556477
EC00237=-270405,-556477
EC00238=-270405,-556477
EC00239=-270405,-556477
EC00240=-270405,-556477
EC00241=-270405,-556477
EC00242=-270405,-556477
EC00243=-270405,-556477
EC00244=-270405,-556477
EC00245=-270405,-556477
EC00246=-270405,-556477
EC00247=-270405,-556477
EC00248=-270405,-556477
EC00249=-270405,-556477
EC00250=-270405,-556477
EC00251=-270405,-556477
EC00252=-270405,-556477
EC00253=-270405,-556477
EC00254=-270405,-556477
EC00255=-270405,-556477
EC00256=-270405,-556477
EC00257=-270405,-556477
EC00258=-270405,-556477
EC00259=-270402,-556478
EC00260=-270402,-556478
EC00261=-270402,-556478
EC00262=-270402,-556478
EC00263=-270402,-556478
EC00264=-270402,-556478
EC00265=-270402,-556478
EC00266=-270402,-556478
EC00267=-270402,-556478
EC00268=-270405,-556477
EC00269=-270405,-556477
EC00270=-270405,-556477
EC00271=-270405,-556477
EC00272=-270405,-556477
EC00273=-270405,-556477
EC00274=-270405,-556477
EC00275=-270405,-556477
EC00276=-270405,-556477
EC00277=-270405,-556477
EC00278=-270405,-556477
EC00279=-270405,-556477
EC00280=-270405,-556477
EC00281=-447795,-556477
EC00282=-447795,-556477
EC00283=-447795,-556477
EC00284=-447795,-556477
EC00285=-447795,-556477
EC00286=-447795,-556477
EC00287=-447795,-556477
EC00288=-447795,-556477
EC00289=-447795,-556477
EC00290=-447795,-556477
EC00291=-447795,-556477
EC00292=-447795,-556477
EC00293=-447795,-556477
EC00294=-447795,-556477
EC00295=-447795,-556477
EC00296=-447795,-556477
EC00297=-447795,-556477
EC00298=-447795,-556477
EC00299=-447795,-556477
EC00300=-447795,-556477
EC00301=-447795,-556477
EC00302=-447795,-556477
EC00303=-447795,-556477
EC00304=-447795,-556477
EC00305=-447795,-556477
EC00306=-447795,-556477
EC00307=-447793,-556477
EC00308=-447793,-556477
EC00309=-447793,-556477
EC00310=-447793,-556477
EC00311=-447793,-556477
EC00312=-447793,-556477
EC00313=-447791,-556477
EC00314=-447791,-556477
EC00315=-447791,-556477
EC00316=-447791,-556477
EC00317=-447791,-556477
EC00318=-447791,-556477
EC00319=-447791,-556477
EC00320=-447791,-556477
EC00321=-447791,-556477
EC00322=-447791,-556477
EC00323=-447791,-556477
EC00324=-447791,-556477
EC00325=-447791,-556477
EC00326=-447791,-556477
EC00327=-447791,-556477
EC00328=-447791,-556477
EC00329=-447791,-556477
EC00330=-447791,-556477
EC00331=-447791,-556477
EC00332=-447791,-556477
EC00333=-447791,-556477
EC00334=-447791,-556477
EC00335=-447791,-556477
EC00336=-447791,-556477
EC00337=-447791,-556477
EC00338=-447791,-556477
EC00339=-447791,-556477
EC00340=-447791,-556477
EC00341=-447791,-556477
EC00342=-447791,-556477
EC00343=-447791,-556477
EC00344=-447791,-556477
EC00345=-447791,-556477
EC00346=-447791,-556477
EC00347=-333615,-556477
EC00348=-311064,-556477
EC00349=-272209,-556477
EC00350=-270405,-556477
EC00351=-270405,-556477
EC00352=-270405,-556477
EC00353=-270405,-556477
EC00354=-270405,-556477
EC00355=-270405,-556477
EC00356=-270405,-556477
EC00357=-270405,-556477
EC00358=-270405,-556477
EC00359=-270405,-556477
EC00360=-270405,-556477
EC00361=-270405,-556477
EC00362=-270405,-556477
EC00363=-270405,-556477
EC00364=-447795,-556477
EC00365=-447795,-556477
EC00366=-447795,-556477
EC00367=-447795,-556477
EC00368=-447795,-556477
EC00369=-447795,-556477
EC00370=-447795,-556477
EC00371=-447795,-556477
EC00372=-447795,-556477
EC00373=-447795,-556477
EC00374=-447795,-556477
EC00375=-447795,-556477
EC00376=-447795,-556477
EC00377=-447795,-556477
EC00378=-447795,-556477
EC00379=-447795,-556477
EC00380=-447795,-556477
EC00381=-447794,-556477
EC00382=-447795,-556477
EC00383=-447795,-556477
EC00384=-447795,-556477
EC00385=-447794,-556478
EC00386=-447795,-556477
EC00387=-447795,-556477
EC00388=-447795,-556477
EC00389=-447795,-556477
EC00390=-447795,-556477
EC00391=-447795,-556477
EC00392=-447795,-556477
EC00393=-447793,-556477
EC00394=-447795,-556477
EC00395=-447795,-556477
EC00396=-447795,-556477
EC00397=-447795,-556477
EC00398=-447795,-556477
EC00399=-447795,-556477
EC00400=-447795,-556477
EC00401=-447795,-556477
EC00402=-447794,-556478
EC00403=-447795,-556477
EC00404=-447795,-556477
EC00405=-447795,-556477
EC00406=-447795,-556477
EC00407=-447795,-556477
EC00408=-447795,-556477
EC00409=-447795,-556477
EC00410=-447795,-556477
EC00411=-447795,-556477
EC00412=-447795,-556477
EC00413=-447795,-556477
EC00414=-71624,-556477
EC00415=15446,-556477
///POSTYPE BASE
///RECTAN
///RCONF 0,0,0,0,0,0,0,0,0,0,0,0,0,0,0,0,0,0,0,0,0,0,0,0
P00006=0.222,-3.123,-1.508,0.0000,0.0000,0.0000
P00032=1.957,0.503,-7.217,0.0000,0.0000,0.0000
///RCONF 0,0,0,0,1,0,0,0,0,0,0,0,0,0,0,0,0,0,0,0,0,0,0,0
P00033=-0.123,0.612,-5.012,0.0000,0.0000,0.0000
///RCONF 0,0,0,0,0,0,0,0,0,0,0,0,0,0,0,0,0,0,0,0,0,0,0,0
P00034=-0.304,0.773,-2.693,0.0000,0.0000,0.0000
P00035=2.817,0.591,-1.622,0.0000,0.0000,0.0000
P00040=-0.030,9.648,2.467,0.0000,0.0000,0.0000
P00041=0.192,3.924,0.305,0.0000,0.0000,0.0000
P00042=-0.217,1.941,0.413,0.0000,0.0000,0.0000
P00043=-0.044,-1.937,1.197,0.0000,0.0000,0.0000
P00044=0.687,-2.322,1.156,0.0000,0.0000,0.0000
P00045=-0.068,-0.810,1.603,0.0000,0.0000,0.0000
P00046=0.799,0.043,1.292,0.0000,0.0000,0.0000
P00048=2.411,0.025,-0.606,0.0000,0.0000,0.0000
P00049=3.413,-3.572,-1.618,0.0000,0.0000,0.0000
P00050=4.296,-4.501,-0.826,0.0000,0.0000,0.0000
//INST
///DATE 2025/03/06 11:55
///ATTR SC,RW
///GROUP1 RB1,BS1
///GROUP2 ST1
NOP
MOVJ C00000 BC00000 VJ=100.00  +MOVJ EC00000 VJ=100.00
MOVJ C00001 BC00001 VJ=100.00  +MOVJ EC00001 VJ=100.00
CALL JOB:CLEAN-R1_KM_NEW
MOVJ C00002 BC00002 VJ=100.00  +MOVJ EC00002 VJ=100.00
MOVJ C00003 BC00003 VJ=50.00  +MOVJ EC00003 VJ=50.00
SMOVL C00004 BC00004 V=83.3  +MOVJ EC00004
SREFP 3 C00005 BC00005  +REFP EC00005
CALL JOB:SEARCH-R1-S13D
SET P032 P006
SFTON3D P032
SMOVL C00006 BC00006 V=60.0  +MOVJ EC00006
SMOVL C00007 BC00007 V=133.3  +MOVJ EC00007
SMOVL C00008 BC00008 V=133.3  +MOVJ EC00008
SREFP 3 C00009 BC00009  +REFP EC00009
CALL JOB:SEARCH-R1-S13D
SET P032 P006
SFTON3D P032
SMOVL C00010 BC00010 V=60.0  +MOVJ EC00010
SMOVL C00011 BC00011 V=133.3  +MOVJ EC00011
SMOVL C00012 BC00012 V=133.3  +MOVJ EC00012
SREFP 3 C00013 BC00013  +REFP EC00013
CALL JOB:SEARCH-R1-S13D
SET P032 P006
SFTON3D P032
SFTOF3D
SMOVL C00014 BC00014 V=133.3  +MOVJ EC00014
SMOVL C00015 BC00015 V=200.0  +MOVJ EC00015
SFTOF3D
'S1
MOVJ C00016 BC00016 VJ=50.00  +MOVJ EC00016 VJ=50.00
'S2
SMOVL C00017 BC00017 V=60.0  +MOVJ EC00017
SREFP 3 C00018 BC00018  +REFP EC00018
CALL JOB:SEARCH-R1-S13D
SET P033 P006
SFTON3D P033
SMOVL C00019 BC00019 V=60.0  +MOVJ EC00019
SMOVL C00020 BC00020 V=133.3  +MOVJ EC00020
SMOVL C00021 BC00021 V=133.3  +MOVJ EC00021
SREFP 3 C00022 BC00022  +REFP EC00022
CALL JOB:SEARCH-R1-S13D
SET P033 P006
SFTON3D P033
SFTOF3D
SMOVL C00023 BC00023 V=83.3  +MOVJ EC00023
MOVJ C00024 BC00024 VJ=60.00  +MOVJ EC00024 VJ=60.00
MOVJ C00025 BC00025 VJ=60.00  +MOVJ EC00025 VJ=60.00
MOVJ C00026 BC00026 VJ=100.00  +MOVJ EC00026 VJ=60.00
MOVJ C00027 BC00027 VJ=60.00  +MOVJ EC00027 VJ=60.00
SMOVL C00028 BC00028 V=60.0  +MOVJ EC00028
SREFP 3 C00029 BC00029  +REFP EC00029
CALL JOB:SEARCH-R1-S13D
SET P034 P006
SFTON3D P034
SMOVL C00030 BC00030 V=60.0  +MOVJ EC00030
SMOVL C00031 BC00031 V=83.3  +MOVJ EC00031
SMOVL C00032 BC00032 V=83.3  +MOVJ EC00032
SREFP 3 C00033 BC00033  +REFP EC00033
CALL JOB:SEARCH-R1-S13D
SET P034 P006
SFTON3D P034
SMOVL C00034 BC00034 V=100.0  +MOVJ EC00034
SMOVL C00035 BC00035 V=133.3  +MOVJ EC00035
SMOVL C00036 BC00036 V=133.3  +MOVJ EC00036
SREFP 3 C00037 BC00037  +REFP EC00037
CALL JOB:SEARCH-R1-S13D
SET P034 P006
SFTON3D P034
SMOVL C00038 BC00038 V=133.3  +MOVJ EC00038
SMOVL C00039 BC00039 V=133.3  +MOVJ EC00039
SMOVL C00040 BC00040 V=250.0  +MOVJ EC00040
SMOVL C00041 BC00041 V=60.0  +MOVJ EC00041
SREFP 3 C00042 BC00042  +REFP EC00042
CALL JOB:SEARCH-R1-S13D
SET P035 P006
SFTON3D P035
SMOVL C00043 BC00043 V=60.0  +MOVJ EC00043
SMOVL C00044 BC00044 V=250.0  +MOVJ EC00044
SMOVL C00045 BC00045 V=250.0  +MOVJ EC00045
SREFP 3 C00046 BC00046  +REFP EC00046
CALL JOB:SEARCH-R1-S13D
SET P035 P006
SFTON3D P035
SMOVL C00047 BC00047 V=166.7  +MOVJ EC00047
SFTOF3D
MOVJ C00048 BC00048 VJ=30.00  +MOVJ EC00048 VJ=15.00
MOVJ C00049 BC00049 VJ=100.00  +MOVJ EC00049 VJ=50.00
MACRO1 MJ#(0) ARGF9
MOVJ C00050 BC00050 VJ=100.00  +MOVJ EC00050 VJ=15.00
SMOVL C00051 BC00051 V=666.7  +MOVJ EC00051
SFTON3D P035
SMOVL C00052 BC00052 V=166.7  +MOVJ EC00052
ARCON
SMOVL C00053 BC00053 V=6.7  +MOVJ EC00053
SMOVL C00054 BC00054 V=6.7  +MOVJ EC00054
ARCOF
TIMER T=1.00
SMOVL C00055 BC00055 V=166.7  +MOVJ EC00055
SFTOF3D
MOVJ C00056 BC00056 VJ=100.00  +MOVJ EC00056 VJ=100.00
MOVJ C00057 BC00057 VJ=15.00  +MOVJ EC00057 VJ=100.00
SFTON3D P035
SMOVL C00058 BC00058 V=166.7  +MOVJ EC00058
ARCON
SFTON3D P034
SMOVL C00059 BC00059 V=8.3  +MOVJ EC00059
SMOVL C00060 BC00060 V=8.3  +MOVJ EC00060
ARCOF
SMOVL C00061 BC00061 V=166.7  +MOVJ EC00061
SMOVL C00062 BC00062 V=500.0  +MOVJ EC00062
SMOVL C00063 BC00063 V=166.7  +MOVJ EC00063
ARCON
SMOVL C00064 BC00064 V=7.5  +MOVJ EC00064
SMOVL C00065 BC00065 V=7.5  +MOVJ EC00065
ARCOF
SFTOF3D
MOVJ C00066 BC00066 VJ=30.00  +MOVJ EC00066 VJ=60.00
MOVJ C00067 BC00067 VJ=100.00  +MOVJ EC00067 VJ=50.00
MOVJ C00068 BC00068 VJ=100.00  +MOVJ EC00068 VJ=15.00
MOVJ C00069 BC00069 VJ=100.00  +MOVJ EC00069 VJ=100.00
MOVJ C00070 BC00070 VJ=50.00  +MOVJ EC00070 VJ=50.00
SFTOF3D
MOVJ C00071 BC00071 VJ=100.00  +MOVJ EC00071 VJ=100.00
MOVJ C00072 BC00072 VJ=100.00  +MOVJ EC00072 VJ=100.00
SFTON3D P033
SMOVL C00073 BC00073 V=166.7  +MOVJ EC00073
ARCON
SFTON3D P032
SMOVL C00074 BC00074 V=8.3  +MOVJ EC00074
SMOVL C00075 BC00075 V=8.3  +MOVJ EC00075
ARCOF
SMOVL C00076 BC00076 V=166.7  +MOVJ EC00076
SMOVL C00077 BC00077 V=666.7  +MOVJ EC00077
SMOVL C00078 BC00078 V=133.3  +MOVJ EC00078
ARCON
SMOVL C00079 BC00079 V=7.5  +MOVJ EC00079
SMOVL C00080 BC00080 V=7.5  +MOVJ EC00080
ARCOF
SFTOF3D
SMOVL C00081 BC00081 V=133.3  +MOVJ EC00081
MOVJ C00082 BC00082 VJ=50.00  +MOVJ EC00082 VJ=50.00
MOVJ C00083 BC00083 VJ=100.00  +MOVJ EC00083 VJ=100.00
MOVJ C00084 BC00084 VJ=100.00  +MOVJ EC00084 VJ=100.00
SFTON3D P033
SMOVL C00085 BC00085 V=133.3  +MOVJ EC00085
ARCON
SMOVL C00086 BC00086 V=7.5  +MOVJ EC00086
ARCON
SMOVL C00087 BC00087 V=7.5  +MOVJ EC00087
ARCOF
MOVJ C00088 BC00088 VJ=50.00  +MOVJ EC00088 VJ=50.00
MOVJ C00089 BC00089 VJ=100.00  +MOVJ EC00089 VJ=100.00
CALL JOB:CLEAN-R1_KM_NEW
MOVJ C00090 BC00090 VJ=100.00  +MOVJ EC00090 VJ=100.00
MOVJ C00091 BC00091 VJ=100.00  +MOVJ EC00091 VJ=100.00
MOVJ C00092 BC00092 VJ=100.00  +MOVJ EC00092 VJ=100.00
MOVJ C00093 BC00093 VJ=100.00  +MOVJ EC00093 VJ=50.00
MOVJ C00094 BC00094 VJ=100.00  +MOVJ EC00094 VJ=50.00
MOVJ C00095 BC00095 VJ=100.00  +MOVJ EC00095 VJ=50.00
MOVJ C00096 BC00096 VJ=100.00  +MOVJ EC00096 VJ=50.00
MOVJ C00097 BC00097 VJ=100.00  +MOVJ EC00097 VJ=15.00
SFTOF3D
MOVJ C00098 BC00098 VJ=15.00  +MOVJ EC00098 VJ=15.00
SMOVL C00099 BC00099 V=100.0  +MOVJ EC00099
SREFP 3 C00100 BC00100  +REFP EC00100
CALL JOB:SEARCH-R1-S13D
SET P041 P006
SFTON3D P041
SMOVL C00101 BC00101 V=100.0  +MOVJ EC00101
SMOVL C00102 BC00102 V=83.3  +MOVJ EC00102
SMOVL C00103 BC00103 V=83.3  +MOVJ EC00103
SREFP 3 C00104 BC00104  +REFP EC00104
CALL JOB:SEARCH-R1-S13D
SET P041 P006
SFTON3D P041
SMOVL C00105 BC00105 V=100.0  +MOVJ EC00105
SFTOF3D
MOVJ C00106 BC00106 VJ=40.00  +MOVJ EC00106 VJ=100.00
MOVJ C00107 BC00107 VJ=100.00  +MOVJ EC00107 VJ=15.00
MOVJ C00108 BC00108 VJ=100.00  +MOVJ EC00108 VJ=15.00
MOVJ C00109 BC00109 VJ=100.00  +MOVJ EC00109 VJ=15.00
MOVJ C00110 BC00110 VJ=100.00  +MOVJ EC00110 VJ=15.00
MOVJ C00111 BC00111 VJ=30.00  +MOVJ EC00111 VJ=15.00
MOVJ C00112 BC00112 VJ=100.00  +MOVJ EC00112 VJ=50.00
MOVJ C00113 BC00113 VJ=50.00  +MOVJ EC00113 VJ=50.00
MOVJ C00114 BC00114 VJ=50.00  +MOVJ EC00114 VJ=50.00
MOVJ C00115 BC00115 VJ=50.00  +MOVJ EC00115 VJ=50.00
MOVJ C00116 BC00116 VJ=50.00  +MOVJ EC00116 VJ=50.00
SFTOF3D
SMOVL C00117 BC00117 V=83.3  +MOVJ EC00117
SREFP 3 C00118 BC00118  +REFP EC00118
CALL JOB:SEARCH-R1-S13D
SET P040 P006
SFTON3D P040
SMOVL C00119 BC00119 V=100.0  +MOVJ EC00119
SMOVL C00120 BC00120 V=133.3  +MOVJ EC00120
SMOVL C00121 BC00121 V=83.3 PL=0  +MOVJ EC00121
SREFP 3 C00122 BC00122  +REFP EC00122
CALL JOB:SEARCH-R1-S13D
SET P040 P006
SFTON3D P040
SMOVL C00123 BC00123 V=100.0  +MOVJ EC00123
SFTOF3D
MACRO1 MJ#(0) ARGF9
SFTON3D P040
SMOVL C00124 BC00124 V=133.3  +MOVJ EC00124
ARCON
SMOVL C00125 BC00125 V=11.7  +MOVJ EC00125
ARCOF
MOVJ C00126 BC00126 VJ=20.00  +MOVJ EC00126 VJ=15.00
MOVJ C00127 BC00127 VJ=30.00  +MOVJ EC00127 VJ=15.00
'SPAWDZIC CZY SPOINA TRAFIA
SMOVL C00128 BC00128 V=166.7  +MOVJ EC00128
ARCON
SMOVL C00129 BC00129 V=12.5  +MOVJ EC00129
ARCOF
SMOVL C00130 BC00130 V=333.3  +MOVJ EC00130
MOVJ C00131 BC00131 VJ=50.00  +MOVJ EC00131 VJ=50.00
MOVJ C00132 BC00132 VJ=100.00  +MOVJ EC00132 VJ=50.00
MOVJ C00133 BC00133 VJ=100.00  +MOVJ EC00133 VJ=50.00
MOVJ C00134 BC00134 VJ=100.00  +MOVJ EC00134 VJ=50.00
SFTON3D P040
SMOVL C00135 BC00135 V=250.0  +MOVJ EC00135
ARCON
SMOVL C00136 BC00136 V=11.7  +MOVJ EC00136
ARCOF
SFTOF3D
MOVJ C00137 BC00137 VJ=25.00  +MOVJ EC00137 VJ=50.00
MOVJ C00138 BC00138 VJ=100.00  +MOVJ EC00138 VJ=50.00
MOVJ C00139 BC00139 VJ=100.00  +MOVJ EC00139 VJ=50.00
MOVJ C00140 BC00140 VJ=100.00  +MOVJ EC00140 VJ=50.00
MOVJ C00141 BC00141 VJ=100.00  +MOVJ EC00141 VJ=50.00
MOVJ C00142 BC00142 VJ=100.00  +MOVJ EC00142 VJ=50.00
SFTOF3D
MOVJ C00143 BC00143 VJ=100.00  +MOVJ EC00143 VJ=50.00
SFTOF3D
MOVJ C00144 BC00144 VJ=100.00  +MOVJ EC00144 VJ=50.00
SFTON3D P041
SMOVL C00145 BC00145 V=200.0  +MOVJ EC00145
ARCON
SMOVL C00146 BC00146 V=10.8  +MOVJ EC00146
ARCOF
SMOVL C00147 BC00147 V=83.3  +MOVJ EC00147
ARCON
SMOVL C00148 BC00148 V=10.0  +MOVJ EC00148
ARCOF
SMOVL C00149 BC00149 V=250.0  +MOVJ EC00149
MOVJ C00150 BC00150 VJ=50.00  +MOVJ EC00150 VJ=50.00
MOVJ C00151 BC00151 VJ=15.00  +MOVJ EC00151 VJ=50.00
SMOVL C00152 BC00152 V=250.0  +MOVJ EC00152
MACRO1 MJ#(0) ARGF9
SMOVL C00153 BC00153 V=200.0  +MOVJ EC00153
ARCON
SMOVL C00154 BC00154 V=11.7  +MOVJ EC00154
ARCOF
SMOVL C00155 BC00155 V=333.3  +MOVJ EC00155
SFTOF3D
MOVJ C00156 BC00156 VJ=100.00  +MOVJ EC00156 VJ=50.00
MOVJ C00157 BC00157 VJ=100.00  +MOVJ EC00157 VJ=50.00
MOVJ C00158 BC00158 VJ=100.00  +MOVJ EC00158 VJ=50.00
MOVJ C00159 BC00159 VJ=100.00  +MOVJ EC00159 VJ=50.00
MOVJ C00160 BC00160 VJ=100.00  +MOVJ EC00160 VJ=50.00
MOVJ C00161 BC00161 VJ=100.00  +MOVJ EC00161 VJ=50.00
MOVJ C00162 BC00162 VJ=100.00  +MOVJ EC00162 VJ=50.00
MOVJ C00163 BC00163 VJ=20.00  +MOVJ EC00163 VJ=50.00
SFTON3D P040
SMOVL C00164 BC00164 V=83.3  +MOVJ EC00164
ARCON
SMOVL C00165 BC00165 V=11.7  +MOVJ EC00165
ARCOF
SMOVL C00166 BC00166 V=133.3  +MOVJ EC00166
SFTOF3D
MOVJ C00167 BC00167 VJ=50.00  +MOVJ EC00167 VJ=50.00
MOVJ C00168 BC00168 VJ=100.00  +MOVJ EC00168 VJ=50.00
MOVJ C00169 BC00169 VJ=100.00  +MOVJ EC00169 VJ=50.00
MOVJ C00170 BC00170 VJ=100.00  +MOVJ EC00170 VJ=50.00
MOVJ C00171 BC00171 VJ=100.00  +MOVJ EC00171 VJ=50.00
MOVJ C00172 BC00172 VJ=100.00  +MOVJ EC00172 VJ=50.00
MOVJ C00173 BC00173 VJ=100.00  +MOVJ EC00173 VJ=50.00
MOVJ C00174 BC00174 VJ=100.00  +MOVJ EC00174 VJ=50.00
MOVJ C00175 BC00175 VJ=15.00  +MOVJ EC00175 VJ=50.00
SFTON3D P041
SMOVL C00176 BC00176 V=133.3  +MOVJ EC00176
ARCON
SMOVL C00177 BC00177 V=11.7  +MOVJ EC00177
ARCOF
SMOVL C00178 BC00178 V=133.3  +MOVJ EC00178
SFTOF3D
MOVJ C00179 BC00179 VJ=100.00  +MOVJ EC00179 VJ=50.00
MOVJ C00180 BC00180 VJ=100.00  +MOVJ EC00180 VJ=50.00
MOVJ C00181 BC00181 VJ=100.00  +MOVJ EC00181 VJ=50.00
MOVJ C00182 BC00182 VJ=100.00  +MOVJ EC00182 VJ=50.00
MOVJ C00183 BC00183 VJ=100.00  +MOVJ EC00183 VJ=50.00
MOVJ C00184 BC00184 VJ=100.00  +MOVJ EC00184 VJ=50.00
MOVJ C00185 BC00185 VJ=100.00  +MOVJ EC00185 VJ=50.00
MOVJ C00186 BC00186 VJ=100.00  +MOVJ EC00186 VJ=50.00
MOVJ C00187 BC00187 VJ=15.00  +MOVJ EC00187 VJ=50.00
SFTON3D P040
SMOVL C00188 BC00188 V=133.3  +MOVJ EC00188
ARCON
SMOVL C00189 BC00189 V=11.7  +MOVJ EC00189
ARCOF
SMOVL C00190 BC00190 V=133.3  +MOVJ EC00190
MOVJ C00191 BC00191 VJ=100.00  +MOVJ EC00191 VJ=50.00
MOVJ C00192 BC00192 VJ=100.00  +MOVJ EC00192 VJ=50.00
MOVJ C00193 BC00193 VJ=100.00  +MOVJ EC00193 VJ=50.00
MOVJ C00194 BC00194 VJ=15.00  +MOVJ EC00194 VJ=15.00
SMOVL C00195 BC00195 V=133.3  +MOVJ EC00195
ARCON
SMOVL C00196 BC00196 V=11.7  +MOVJ EC00196
ARCOF
SMOVL C00197 BC00197 V=133.3  +MOVJ EC00197
SMOVL C00198 BC00198 V=133.3  +MOVJ EC00198
ARCON
SMOVL C00199 BC00199 V=11.7  +MOVJ EC00199
ARCOF
SFTOF3D
SMOVL C00200 BC00200 V=133.3  +MOVJ EC00200
MOVJ C00201 BC00201 VJ=100.00  +MOVJ EC00201 VJ=50.00
MOVJ C00202 BC00202 VJ=100.00  +MOVJ EC00202 VJ=50.00
MOVJ C00203 BC00203 VJ=100.00  +MOVJ EC00203 VJ=50.00
MOVJ C00204 BC00204 VJ=100.00  +MOVJ EC00204 VJ=50.00
MOVJ C00205 BC00205 VJ=100.00  +MOVJ EC00205 VJ=50.00
MOVJ C00206 BC00206 VJ=100.00  +MOVJ EC00206 VJ=50.00
MOVJ C00207 BC00207 VJ=100.00  +MOVJ EC00207 VJ=50.00
MOVJ C00208 BC00208 VJ=100.00  +MOVJ EC00208 VJ=50.00
MOVJ C00209 BC00209 VJ=50.00  +MOVJ EC00209 VJ=50.00
SFTON3D P041
SMOVL C00210 BC00210 V=16.7  +MOVJ EC00210
ARCON
SMOVL C00211 BC00211 V=8.3  +MOVJ EC00211
ARCOF
SMOVL C00212 BC00212 V=250.0  +MOVJ EC00212
MOVJ C00213 BC00213 VJ=100.00  +MOVJ EC00213 VJ=50.00
MACRO1 MJ#(0) ARGF9
SMOVL C00214 BC00214 V=250.0  +MOVJ EC00214
ARCON
SMOVL C00215 BC00215 V=11.7  +MOVJ EC00215
SMOVL C00216 BC00216 V=11.7  +MOVJ EC00216
ARCOF
SMOVL C00217 BC00217 V=166.7  +MOVJ EC00217
SMOVL C00218 BC00218 V=666.7  +MOVJ EC00218
SMOVL C00219 BC00219 V=250.0  +MOVJ EC00219
ARCON
SMOVL C00220 BC00220 V=11.7  +MOVJ EC00220
ARCOF
SFTOF3D
SMOVL C00221 BC00221 V=166.7  +MOVJ EC00221
MOVJ C00222 BC00222 VJ=100.00  +MOVJ EC00222 VJ=50.00
MOVJ C00223 BC00223 VJ=100.00  +MOVJ EC00223 VJ=50.00
MOVJ C00224 BC00224 VJ=100.00  +MOVJ EC00224 VJ=50.00
MOVJ C00225 BC00225 VJ=100.00  +MOVJ EC00225 VJ=50.00
MOVJ C00226 BC00226 VJ=100.00  +MOVJ EC00226 VJ=50.00
MOVJ C00227 BC00227 VJ=50.00  +MOVJ EC00227 VJ=50.00
MOVJ C00228 BC00228 VJ=50.00  +MOVJ EC00228 VJ=50.00
MOVJ C00229 BC00229 VJ=50.00  +MOVJ EC00229 VJ=50.00
SFTON3D P040
SMOVL C00230 BC00230 V=166.7  +MOVJ EC00230
ARCON
SMOVL C00231 BC00231 V=11.7  +MOVJ EC00231
ARCOF
SMOVL C00232 BC00232 V=333.3  +MOVJ EC00232
SMOVL C00233 BC00233 V=666.7  +MOVJ EC00233
SMOVL C00234 BC00234 V=166.7  +MOVJ EC00234
ARCON
SMOVL C00235 BC00235 V=11.7  +MOVJ EC00235
ARCOF
SMOVL C00236 BC00236 V=333.3  +MOVJ EC00236
SFTOF3D
MOVJ C00237 BC00237 VJ=50.00  +MOVJ EC00237 VJ=50.00
MOVJ C00238 BC00238 VJ=50.00  +MOVJ EC00238 VJ=50.00
MOVJ C00239 BC00239 VJ=50.00  +MOVJ EC00239 VJ=50.00
MOVJ C00240 BC00240 VJ=50.00  +MOVJ EC00240 VJ=50.00
MOVJ C00241 BC00241 VJ=50.00  +MOVJ EC00241 VJ=50.00
MOVJ C00242 BC00242 VJ=100.00  +MOVJ EC00242 VJ=50.00
MOVJ C00243 BC00243 VJ=100.00  +MOVJ EC00243 VJ=50.00
MOVJ C00244 BC00244 VJ=50.00  +MOVJ EC00244 VJ=50.00
SFTON3D P041
SMOVL C00245 BC00245 V=250.0  +MOVJ EC00245
ARCON
SMOVL C00246 BC00246 V=11.7  +MOVJ EC00246
ARCOF
SMOVL C00247 BC00247 V=250.0  +MOVJ EC00247
SMOVL C00248 BC00248 V=250.0  +MOVJ EC00248
ARCON
SMOVL C00249 BC00249 V=10.8  +MOVJ EC00249
ARCOF
SMOVL C00250 BC00250 V=250.0  +MOVJ EC00250
SMOVL C00251 BC00251 V=666.7  +MOVJ EC00251
MOVJ C00252 BC00252 VJ=100.00  +MOVJ EC00252 VJ=50.00
SSFTOF
MOVJ C00253 BC00253 VJ=100.00  +MOVJ EC00253 VJ=50.00
CALL JOB:CLEAN-R1_KM2
MOVJ C00254 BC00254 VJ=100.00  +MOVJ EC00254 VJ=50.00
MOVJ C00255 BC00255 VJ=100.00  +MOVJ EC00255 VJ=15.00
MOVJ C00256 BC00256 VJ=100.00  +MOVJ EC00256 VJ=50.00
MOVJ C00257 BC00257 VJ=100.00  +MOVJ EC00257 VJ=50.00
MOVJ C00258 BC00258 VJ=15.00  +MOVJ EC00258 VJ=15.00
MOVJ C00259 BC00259 VJ=15.00  +MOVJ EC00259 VJ=50.00
SMOVL C00260 BC00260 V=83.3  +MOVJ EC00260
SREFP 3 C00261 BC00261  +REFP EC00261
CALL JOB:SEARCH-R1-S13D
SET P042 P006
SFTON3D P042
SMOVL C00262 BC00262 V=60.0  +MOVJ EC00262
SMOVL C00263 BC00263 V=133.3  +MOVJ EC00263
SMOVL C00264 BC00264 V=133.3  +MOVJ EC00264
SREFP 3 C00265 BC00265  +REFP EC00265
CALL JOB:SEARCH-R1-S13D
SET P042 P006
SFTON3D P042
SMOVL C00266 BC00266 V=60.0  +MOVJ EC00266
SFTOF3D
MOVJ C00267 BC00267 VJ=15.00  +MOVJ EC00267 VJ=15.00
MOVJ C00268 BC00268 VJ=15.00  +MOVJ EC00268 VJ=15.00
MOVJ C00269 BC00269 VJ=15.00  +MOVJ EC00269 VJ=15.00
MOVJ C00270 BC00270 VJ=15.00  +MOVJ EC00270 VJ=15.00
SMOVL C00271 BC00271 V=83.3  +MOVJ EC00271
SREFP 3 C00272 BC00272  +REFP EC00272
CALL JOB:SEARCH-R1-S13D
SET P043 P006
SFTON3D P043
SMOVL C00273 BC00273 V=60.0  +MOVJ EC00273
SMOVL C00274 BC00274 V=133.3  +MOVJ EC00274
SMOVL C00275 BC00275 V=133.3  +MOVJ EC00275
SREFP 3 C00276 BC00276  +REFP EC00276
CALL JOB:SEARCH-R1-S13D
SET P043 P006
SFTON3D P043
SMOVL C00277 BC00277 V=60.0  +MOVJ EC00277
MOVJ C00278 BC00278 VJ=30.00  +MOVJ EC00278 VJ=30.00
SFTOF3D
MOVJ C00279 BC00279 VJ=30.00  +MOVJ EC00279 VJ=30.00
MOVJ C00280 BC00280 VJ=30.00  +MOVJ EC00280 VJ=30.00
MOVJ C00281 BC00281 VJ=50.00  +MOVJ EC00281 VJ=50.00
MOVJ C00282 BC00282 VJ=50.00  +MOVJ EC00282 VJ=50.00
SFTOF3D
MOVJ C00283 BC00283 VJ=30.00  +MOVJ EC00283 VJ=30.00
SMOVL C00284 BC00284 V=83.3  +MOVJ EC00284
SREFP 3 C00285 BC00285  +REFP EC00285
CALL JOB:SEARCH-R1-S13D
SET P044 P006
SFTON3D P044
SMOVL C00286 BC00286 V=100.0  +MOVJ EC00286
SREFP 3 C00287 BC00287  +REFP EC00287
CALL JOB:SEARCH-R1-S13D
SET P044 P006
SFTON3D P044
SMOVL C00288 BC00288 V=133.3  +MOVJ EC00288
SMOVL C00289 BC00289 V=250.0  +MOVJ EC00289
SMOVL C00290 BC00290 V=133.3  +MOVJ EC00290
SREFP 3 C00291 BC00291  +REFP EC00291
CALL JOB:SEARCH-R1-S13D
SET P044 P006
SFTON3D P044
SMOVL C00292 BC00292 V=133.3  +MOVJ EC00292
SFTOF3D
MOVJ C00293 BC00293 VJ=30.00  +MOVJ EC00293 VJ=15.00
MOVJ C00294 BC00294 VJ=30.00  +MOVJ EC00294 VJ=15.00
MOVJ C00295 BC00295 VJ=30.00  +MOVJ EC00295 VJ=15.00
SMOVL C00296 BC00296 V=250.0  +MOVJ EC00296
SREFP 3 C00297 BC00297  +REFP EC00297
CALL JOB:SEARCH-R1-S13D
SET P045 P006
SFTON3D P045
SMOVL C00298 BC00298 V=250.0  +MOVJ EC00298
SREFP 3 C00299 BC00299  +REFP EC00299
CALL JOB:SEARCH-R1-S13D
SET P045 P006
SFTON3D P045
SMOVL C00300 BC00300 V=250.0  +MOVJ EC00300
SMOVL C00301 BC00301 V=250.0  +MOVJ EC00301
SMOVL C00302 BC00302 V=166.7  +MOVJ EC00302
SREFP 3 C00303 BC00303  +REFP EC00303
CALL JOB:SEARCH-R1-S13D
SET P045 P006
SFTON3D P045
SMOVL C00304 BC00304 V=250.0  +MOVJ EC00304
SFTOF3D
MOVJ C00305 BC00305 VJ=30.00  +MOVJ EC00305 VJ=15.00
MOVJ C00306 BC00306 VJ=30.00  +MOVJ EC00306 VJ=15.00
SMOVL C00307 BC00307 V=250.0  +MOVJ EC00307
SREFP 3 C00308 BC00308  +REFP EC00308
CALL JOB:SEARCH-R1-S13D
SET P046 P006
SFTON3D P046
SMOVL C00309 BC00309 V=250.0  +MOVJ EC00309
SREFP 3 C00310 BC00310  +REFP EC00310
CALL JOB:SEARCH-R1-S13D
SET P046 P006
SFTON3D P046
SMOVL C00311 BC00311 V=250.0  +MOVJ EC00311
SFTOF3D
MOVJ C00312 BC00312 VJ=30.00  +MOVJ EC00312 VJ=15.00
MOVJ C00313 BC00313 VJ=30.00  +MOVJ EC00313 VJ=15.00
MOVJ C00314 BC00314 VJ=30.00  +MOVJ EC00314 VJ=15.00
MOVJ C00315 BC00315 VJ=30.00  +MOVJ EC00315 VJ=15.00
SMOVL C00316 BC00316 V=250.0  +MOVJ EC00316
SREFP 3 C00317 BC00317  +REFP EC00317
CALL JOB:SEARCH-R1-S13D
SET P048 P006
SFTON3D P048
SMOVL C00318 BC00318 V=250.0  +MOVJ EC00318
SREFP 3 C00319 BC00319  +REFP EC00319
CALL JOB:SEARCH-R1-S13D
SET P048 P006
SFTON3D P048
SMOVL C00320 BC00320 V=250.0  +MOVJ EC00320
MOVJ C00321 BC00321 VJ=30.00  +MOVJ EC00321 VJ=15.00
SFTOF3D
MOVJ C00322 BC00322 VJ=30.00  +MOVJ EC00322 VJ=15.00
MOVJ C00323 BC00323 VJ=30.00  +MOVJ EC00323 VJ=15.00
SMOVL C00324 BC00324 V=166.7  +MOVJ EC00324
SREFP 3 C00325 BC00325  +REFP EC00325
CALL JOB:SEARCH-R1-S13D
SET P049 P006
SFTON3D P049
SMOVL C00326 BC00326 V=166.7  +MOVJ EC00326
SREFP 3 C00327 BC00327  +REFP EC00327
CALL JOB:SEARCH-R1-S13D
SET P049 P006
SFTON3D P049
SMOVL C00328 BC00328 V=166.7  +MOVJ EC00328
SMOVL C00329 BC00329 V=166.7  +MOVJ EC00329
SMOVL C00330 BC00330 V=166.7  +MOVJ EC00330
SREFP 3 C00331 BC00331  +REFP EC00331
CALL JOB:SEARCH-R1-S13D
SET P049 P006
SFTON3D P049
SMOVL C00332 BC00332 V=166.7  +MOVJ EC00332
SFTOF3D
MOVJ C00333 BC00333 VJ=30.00  +MOVJ EC00333 VJ=30.00
MOVJ C00334 BC00334 VJ=30.00  +MOVJ EC00334 VJ=30.00
MOVJ C00335 BC00335 VJ=30.00  +MOVJ EC00335 VJ=15.00
SMOVL C00336 BC00336 V=250.0  +MOVJ EC00336
SREFP 3 C00337 BC00337  +REFP EC00337
CALL JOB:SEARCH-R1-S13D
SET P050 P006
SFTON3D P050
SMOVL C00338 BC00338 V=250.0  +MOVJ EC00338
SREFP 3 C00339 BC00339  +REFP EC00339
CALL JOB:SEARCH-R1-S13D
SET P050 P006
SFTON3D P050
SMOVL C00340 BC00340 V=250.0  +MOVJ EC00340
SMOVL C00341 BC00341 V=250.0  +MOVJ EC00341
SMOVL C00342 BC00342 V=166.7  +MOVJ EC00342
SREFP 3 C00343 BC00343  +REFP EC00343
CALL JOB:SEARCH-R1-S13D
SET P050 P006
SFTON3D P050
SMOVL C00344 BC00344 V=166.7  +MOVJ EC00344
SFTOF3D
MOVJ C00345 BC00345 VJ=30.00  +MOVJ EC00345 VJ=15.00
MOVJ C00346 BC00346 VJ=30.00  +MOVJ EC00346 VJ=15.00
MOVJ C00347 BC00347 VJ=30.00  +MOVJ EC00347 VJ=15.00
MOVJ C00348 BC00348 VJ=30.00  +MOVJ EC00348 VJ=30.00
MOVJ C00349 BC00349 VJ=30.00  +MOVJ EC00349 VJ=30.00
MACRO1 MJ#(0) ARGF9
SFTON3D P042
SMOVL C00350 BC00350 V=166.7  +MOVJ EC00350
ARCON
SMOVC C00351 BC00351 V=8.3  +MOVJ EC00351
SMOVC C00352 BC00352 V=8.3  +MOVJ EC00352
SMOVC C00353 BC00353 V=8.3  +MOVJ EC00353
SMOVL C00354 BC00354 V=8.3  +MOVJ EC00354
ARCOF
SFTOF3D
SMOVL C00355 BC00355 V=250.0  +MOVJ EC00355
SMOVL C00356 BC00356 V=250.0  +MOVJ EC00356
SFTON3D P043
SMOVL C00357 BC00357 V=166.7  +MOVJ EC00357
ARCON
SMOVC C00358 BC00358 V=8.3  +MOVJ EC00358
SMOVC C00359 BC00359 V=8.3  +MOVJ EC00359
SMOVC C00360 BC00360 V=8.3  +MOVJ EC00360
SMOVL C00361 BC00361 V=8.3  +MOVJ EC00361
ARCOF
SFTOF3D
SMOVL C00362 BC00362 V=166.7  +MOVJ EC00362
SMOVL C00363 BC00363 V=250.0  +MOVJ EC00363
MOVJ C00364 BC00364 VJ=30.00  +MOVJ EC00364 VJ=30.00
MACRO1 MJ#(0) ARGF9
MOVJ C00365 BC00365 VJ=15.00  +MOVJ EC00365 VJ=10.00
SFTON3D P044
SMOVL C00366 BC00366 V=166.7  +MOVJ EC00366
ARCON
SMOVL C00367 BC00367 V=9.2  +MOVJ EC00367
SMOVL C00368 BC00368 V=9.2  +MOVJ EC00368
ARCOF
SFTOF3D
SMOVL C00369 BC00369 V=250.0  +MOVJ EC00369
SFTON3D P045
SMOVL C00370 BC00370 V=166.7  +MOVJ EC00370
ARCON
SMOVL C00371 BC00371 V=9.2  +MOVJ EC00371
SMOVL C00372 BC00372 V=9.2  +MOVJ EC00372
ARCOF
SMOVL C00373 BC00373 V=250.0  +MOVJ EC00373
SFTON3D P046
SMOVL C00374 BC00374 V=166.7  +MOVJ EC00374
ARCON
SMOVL C00375 BC00375 V=9.2  +MOVJ EC00375
SMOVL C00376 BC00376 V=9.2  +MOVJ EC00376
ARCOF
SFTOF3D
SMOVL C00377 BC00377 V=166.7  +MOVJ EC00377
SMOVL C00378 BC00378 V=250.0  +MOVJ EC00378
SMOVL C00379 BC00379 V=250.0  +MOVJ EC00379
SMOVL C00380 BC00380 V=250.0  +MOVJ EC00380
SFTON3D P045
SMOVL C00381 BC00381 V=166.7  +MOVJ EC00381
ARCON
SMOVL C00382 BC00382 V=10.0  +MOVJ EC00382
ARCOF
SMOVL C00383 BC00383 V=250.0  +MOVJ EC00383
SMOVL C00384 BC00384 V=333.3  +MOVJ EC00384
SFTON3D P044
SMOVL C00385 BC00385 V=166.7  +MOVJ EC00385
ARCON
SMOVL C00386 BC00386 V=10.0  +MOVJ EC00386
ARCOF
SMOVL C00387 BC00387 V=250.0  +MOVJ EC00387
MOVJ C00388 BC00388 VJ=20.00  +MOVJ EC00388 VJ=10.00
MOVJ C00389 BC00389 VJ=40.00  +MOVJ EC00389 VJ=10.00
MOVJ C00390 BC00390 VJ=20.00  +MOVJ EC00390 VJ=10.00
SFTON3D P050
SMOVL C00391 BC00391 V=166.7  +MOVJ EC00391
ARCON
SMOVL C00392 BC00392 V=9.2  +MOVJ EC00392
SMOVL C00393 BC00393 V=9.2  +MOVJ EC00393
ARCOF
SMOVL C00394 BC00394 V=166.7  +MOVJ EC00394
SFTON3D P049
SMOVL C00395 BC00395 V=166.7  +MOVJ EC00395
ARCON
SMOVL C00396 BC00396 V=9.2  +MOVJ EC00396
SMOVL C00397 BC00397 V=9.2  +MOVJ EC00397
SMOVL C00398 BC00398 V=9.2  +MOVJ EC00398
ARCOF
SMOVL C00399 BC00399 V=166.7  +MOVJ EC00399
SFTON3D P048
SMOVL C00400 BC00400 V=166.7  +MOVJ EC00400
ARCON
SMOVL C00401 BC00401 V=9.2  +MOVJ EC00401
SMOVL C00402 BC00402 V=9.2  +MOVJ EC00402
SMOVL C00403 BC00403 V=8.3  +MOVJ EC00403
ARCOF
SMOVL C00404 BC00404 V=166.7  +MOVJ EC00404
SMOVL C00405 BC00405 V=166.7  +MOVJ EC00405
SFTON3D P049
SMOVL C00406 BC00406 V=166.7  +MOVJ EC00406
ARCON
SMOVL C00407 BC00407 V=10.0  +MOVJ EC00407
ARCOF
SMOVL C00408 BC00408 V=250.0  +MOVJ EC00408
SFTON3D P050
SMOVL C00409 BC00409 V=200.0  +MOVJ EC00409
ARCON
SMOVL C00410 BC00410 V=10.0  +MOVJ EC00410
ARCOF
SFTOF3D
SMOVL C00411 BC00411 V=250.0  +MOVJ EC00411
MOVJ C00412 BC00412 VJ=60.00  +MOVJ EC00412 VJ=60.00
MOVJ C00413 BC00413 VJ=60.00  +MOVJ EC00413 VJ=60.00
MOVJ C00414 BC00414 VJ=60.00  +MOVJ EC00414 VJ=60.00
MOVJ C00415 BC00415 VJ=100.00  +MOVJ EC00415 VJ=100.00
END
